Fanuc KAREL source: kb00170.KL

-- PROVISIONAL review KL for V770-1; original PC SHA256 3032e0a2cacc9c03d34b46ddb95381deb16c99795b3e235c14e976d34489d791
-- Incomplete behavior may be omitted. Consult companion uncertainty JSON. Do not deploy.
PROGRAM KB00170
%NOLOCKGROUP
BEGIN
  -- UNRESOLVED_PC offsets 5-12; opcodes 9D,23
  -- UNRESOLVED_PC offsets 17-24; opcodes 9D,23
  -- UNRESOLVED_PC offsets 29-36; opcodes 9D,23
  -- UNRESOLVED_PC offsets 41-48; opcodes 9D,23
  -- UNRESOLVED_PC offsets 53-60; opcodes 9D,23
  -- UNRESOLVED_PC offsets 65-72; opcodes 9D,23
  -- UNRESOLVED_PC offsets 77-84; opcodes 9D,23
  -- UNRESOLVED_PC offsets 89-96; opcodes 9D,23
  -- UNRESOLVED_PC offsets 101-153; opcodes 27,22,22,22,22,22,22,22,22,31
  -- UNRESOLVED_PC offsets 158-162; opcodes 7F
END KB00170
